// TIA Portal V20 export
FUNCTION "CallSimulation" : Void   // FC22, LAD
TITLE = CallSimulation
// This blocks switches between simulation with SIMIT and PLCSIM Advanced or with PLCSIM and PLC internal simulation function blocks
// stored: IsIECCheckEnabled true, SetENOAutomatically true
   VAR CONSTANT
      True : Bool := true;   // OEM: replace with ProDiag statuses that command unit state
      False : Bool;
   END_VAR
   VAR_TEMP   // added for the SCL form of the ladder/FBD networks
      _w1 : Bool;
      _w2 : Bool;
      _w3 : Bool;
      _w4 : Bool;
      _w5 : Bool;
   END_VAR
BEGIN

REGION Network 1: SIMIT simulation currently running
   // The input "0.000CC1-KE50_I1.6_SimitRunning" is a life bit from SIMIT, which is always TRUE while SIMIT is running. The following actions are performed in that case:
   // - Simulation button in HMI is not shown when a SIMIT simulation is currently running
   // - Deactivate PLC internal simulation while SIMIT simulation is running
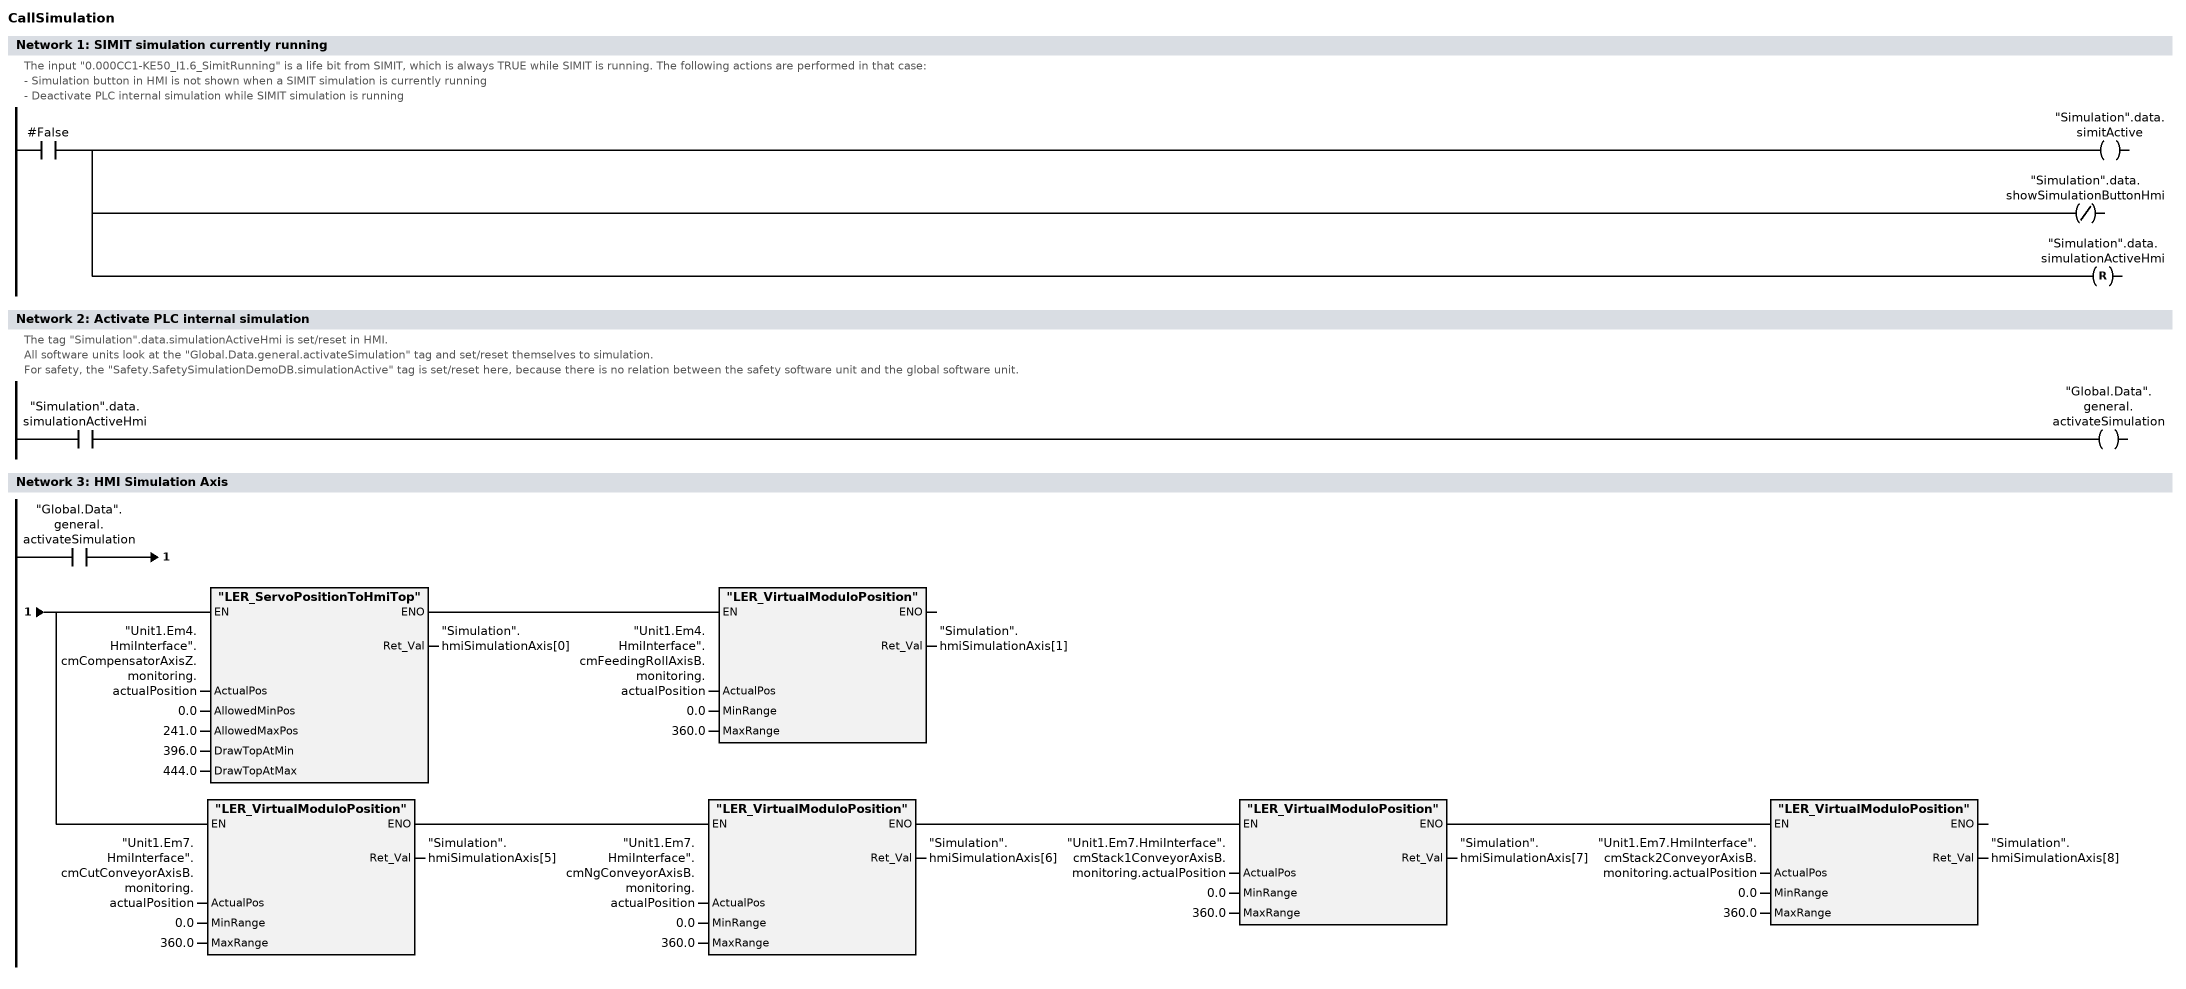
   RUNG wire#powerrail
      Contact( #False )
      wire#w1
      Coil( "Simulation".data.simitActive )
   END_RUNG
   RUNG wire#w1
      I_Coil( "Simulation".data.showSimulationButtonHmi )
   END_RUNG
   RUNG wire#w1
      R_Coil( "Simulation".data.simulationActiveHmi )
   END_RUNG
   // the same network as SCL:
   "Simulation".data.simitActive := #False;
   "Simulation".data.showSimulationButtonHmi := NOT #False;
   IF #False THEN "Simulation".data.simulationActiveHmi := FALSE; END_IF;
END_REGION

REGION Network 2: Activate PLC internal simulation
   // The tag "Simulation".data.simulationActiveHmi is set/reset in HMI.
   // 
   // All software units look at the "Global.Data.general.activateSimulation" tag and set/reset themselves to simulation.
   // 
   // For safety, the "Safety.SafetySimulationDemoDB.simulationActive" tag is set/reset here, because there is no relation between the safety software unit and the global software unit.
   RUNG wire#powerrail
      Contact( "Simulation".data.simulationActiveHmi )
      Coil( "Global.Data".general.activateSimulation )
   END_RUNG
   // the same network as SCL:
   "Global.Data".general.activateSimulation := "Simulation".data.simulationActiveHmi;
END_REGION

REGION Network 3: HMI Simulation Axis
   RUNG wire#powerrail
      Contact( "Global.Data".general.activateSimulation )
      wire#w1
      "LER_ServoPositionToHmiTop"(ActualPos := "Unit1.Em4.HmiInterface".cmCompensatorAxisZ.monitoring.actualPosition, AllowedMinPos := 0.0, AllowedMaxPos := 241.0, DrawTopAtMin := 396.0, DrawTopAtMax := 444.0, Ret_Val => "Simulation".hmiSimulationAxis[0])
      "LER_VirtualModuloPosition"(ActualPos := "Unit1.Em4.HmiInterface".cmFeedingRollAxisB.monitoring.actualPosition, MinRange := 0.0, MaxRange := 360.0, Ret_Val => "Simulation".hmiSimulationAxis[1])
   END_RUNG
   RUNG wire#w1
      "LER_VirtualModuloPosition"(ActualPos := "Unit1.Em7.HmiInterface".cmCutConveyorAxisB.monitoring.actualPosition, MinRange := 0.0, MaxRange := 360.0, Ret_Val => "Simulation".hmiSimulationAxis[5])
      "LER_VirtualModuloPosition"(ActualPos := "Unit1.Em7.HmiInterface".cmNgConveyorAxisB.monitoring.actualPosition, MinRange := 0.0, MaxRange := 360.0, Ret_Val => "Simulation".hmiSimulationAxis[6])
      "LER_VirtualModuloPosition"(ActualPos := "Unit1.Em7.HmiInterface".cmStack1ConveyorAxisB.monitoring.actualPosition, MinRange := 0.0, MaxRange := 360.0, Ret_Val => "Simulation".hmiSimulationAxis[7])
      "LER_VirtualModuloPosition"(ActualPos := "Unit1.Em7.HmiInterface".cmStack2ConveyorAxisB.monitoring.actualPosition, MinRange := 0.0, MaxRange := 360.0, Ret_Val => "Simulation".hmiSimulationAxis[8])
   END_RUNG
   // the same network as SCL:
   #_w2 := "Global.Data".general.activateSimulation;
   "Simulation".hmiSimulationAxis[0] := "LER_ServoPositionToHmiTop"(EN := "Global.Data".general.activateSimulation,
                           ActualPos := "Unit1.Em4.HmiInterface".cmCompensatorAxisZ.monitoring.actualPosition,
                           AllowedMinPos := 0.0,
                           AllowedMaxPos := 241.0,
                           DrawTopAtMin := 396.0,
                           DrawTopAtMax := 444.0,
                           ENO => #_w1);
   IF #_w1 THEN
       "Simulation".hmiSimulationAxis[1] := "LER_VirtualModuloPosition"(ActualPos := "Unit1.Em4.HmiInterface".cmFeedingRollAxisB.monitoring.actualPosition,
                               MinRange := 0.0,
                               MaxRange := 360.0);
   END_IF;
   "Simulation".hmiSimulationAxis[5] := "LER_VirtualModuloPosition"(EN := #_w2,
                           ActualPos := "Unit1.Em7.HmiInterface".cmCutConveyorAxisB.monitoring.actualPosition,
                           MinRange := 0.0,
                           MaxRange := 360.0,
                           ENO => #_w3);
   "Simulation".hmiSimulationAxis[6] := "LER_VirtualModuloPosition"(EN := #_w3,
                           ActualPos := "Unit1.Em7.HmiInterface".cmNgConveyorAxisB.monitoring.actualPosition,
                           MinRange := 0.0,
                           MaxRange := 360.0,
                           ENO => #_w4);
   "Simulation".hmiSimulationAxis[7] := "LER_VirtualModuloPosition"(EN := #_w4,
                           ActualPos := "Unit1.Em7.HmiInterface".cmStack1ConveyorAxisB.monitoring.actualPosition,
                           MinRange := 0.0,
                           MaxRange := 360.0,
                           ENO => #_w5);
   IF #_w5 THEN
       "Simulation".hmiSimulationAxis[8] := "LER_VirtualModuloPosition"(ActualPos := "Unit1.Em7.HmiInterface".cmStack2ConveyorAxisB.monitoring.actualPosition,
                               MinRange := 0.0,
                               MaxRange := 360.0);
   END_IF;
END_REGION
END_FUNCTION
